// Mitsubishi GX Works2 project: 20190826   PLC: FX3U/FX3UC

PROGRAM MAIN
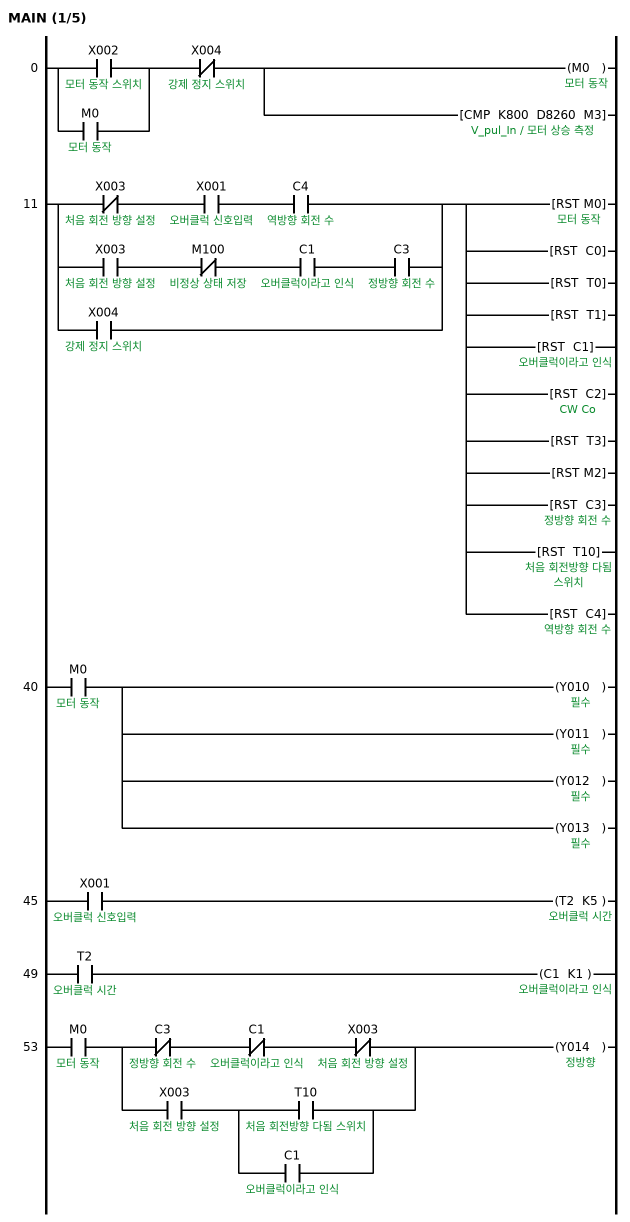
0     LD      X002  ; 모터 동작 스위치
      OR      M0  ; 모터 동작
      ANI     X004  ; 강제 정지 스위치
      OUT     M0  ; 모터 동작
      CMP     K800 D8260 M3  ; V_pul_In / 모터 상승 측정
11    LDI     X003  ; 처음 회전 방향 설정
      AND     X001  ; 오버클럭 신호입력
      AND     C4  ; 역방향 회전 수
      LD      X003  ; 처음 회전 방향 설정
      ANI     M100  ; 비정상 상태 저장
      AND     C1  ; 오버클럭이라고 인식
      AND     C3  ; 정방향 회전 수
      ORB
      OR      X004  ; 강제 정지 스위치
      RST     M0  ; 모터 동작
      RST     C0
      RST     T0
      RST     T1
      RST     C1  ; 오버클럭이라고 인식
      RST     C2  ; CW Co
      RST     T3
      RST     M2
      RST     C3  ; 정방향 회전 수
      RST     T10  ; 처음 회전방향 다됨 스위치
      RST     C4  ; 역방향 회전 수
40    LD      M0  ; 모터 동작
      OUT     Y010  ; 필수
      OUT     Y011  ; 필수
      OUT     Y012  ; 필수
      OUT     Y013  ; 필수
45    LD      X001  ; 오버클럭 신호입력
      OUT     T2 K5  ; 오버클럭 시간
49    LD      T2  ; 오버클럭 시간
      OUT     C1 K1  ; 오버클럭이라고 인식
53    LD      M0  ; 모터 동작
      LDI     C3  ; 정방향 회전 수
      ANI     C1  ; 오버클럭이라고 인식
      ANI     X003  ; 처음 회전 방향 설정
      LD      X003  ; 처음 회전 방향 설정
      LD      T10  ; 처음 회전방향 다됨 스위치
      OR      C1  ; 오버클럭이라고 인식
      ANB
      ORB
      ANB
      OUT     Y014  ; 정방향
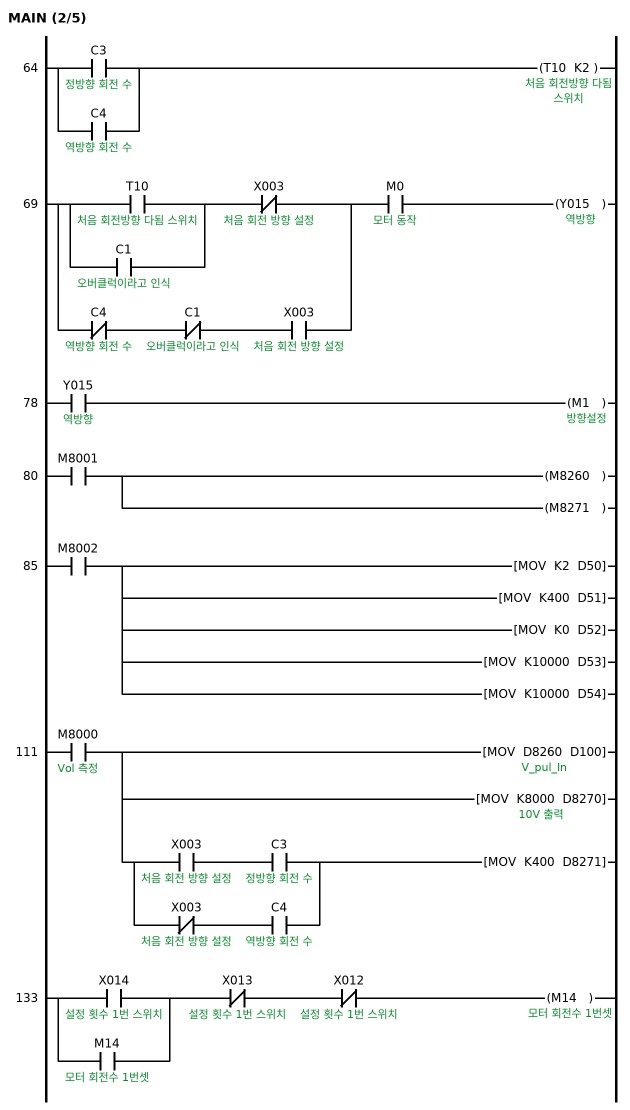
64    LD      C3  ; 정방향 회전 수
      OR      C4  ; 역방향 회전 수
      OUT     T10 K2  ; 처음 회전방향 다됨 스위치
69    LD      T10  ; 처음 회전방향 다됨 스위치
      OR      C1  ; 오버클럭이라고 인식
      ANI     X003  ; 처음 회전 방향 설정
      LDI     C4  ; 역방향 회전 수
      ANI     C1  ; 오버클럭이라고 인식
      AND     X003  ; 처음 회전 방향 설정
      ORB
      AND     M0  ; 모터 동작
      OUT     Y015  ; 역방향
78    LD      Y015  ; 역방향
      OUT     M1  ; 방향설정
80    LD      M8001
      OUT     M8260
      OUT     M8271
85    LD      M8002
      MOV     K2 D50
      MOV     K400 D51
      MOV     K0 D52
      MOV     K10000 D53
      MOV     K10000 D54
111   LD      M8000  ; Vol 측정
      MOV     D8260 D100
      MOV     K8000 D8270  ; 10V 출력
      LD      X003  ; 처음 회전 방향 설정
      AND     C3  ; 정방향 회전 수
      LDI     X003  ; 처음 회전 방향 설정
      AND     C4  ; 역방향 회전 수
      ORB
      ANB
      MOV     K400 D8271
133   LD      X014  ; 설정 횟수 1번 스위치
      OR      M14  ; 모터 회전수 1번셋
      ANI     X013  ; 설정 횟수 1번 스위치
      ANI     X012  ; 설정 횟수 1번 스위치
      OUT     M14  ; 모터 회전수 1번셋
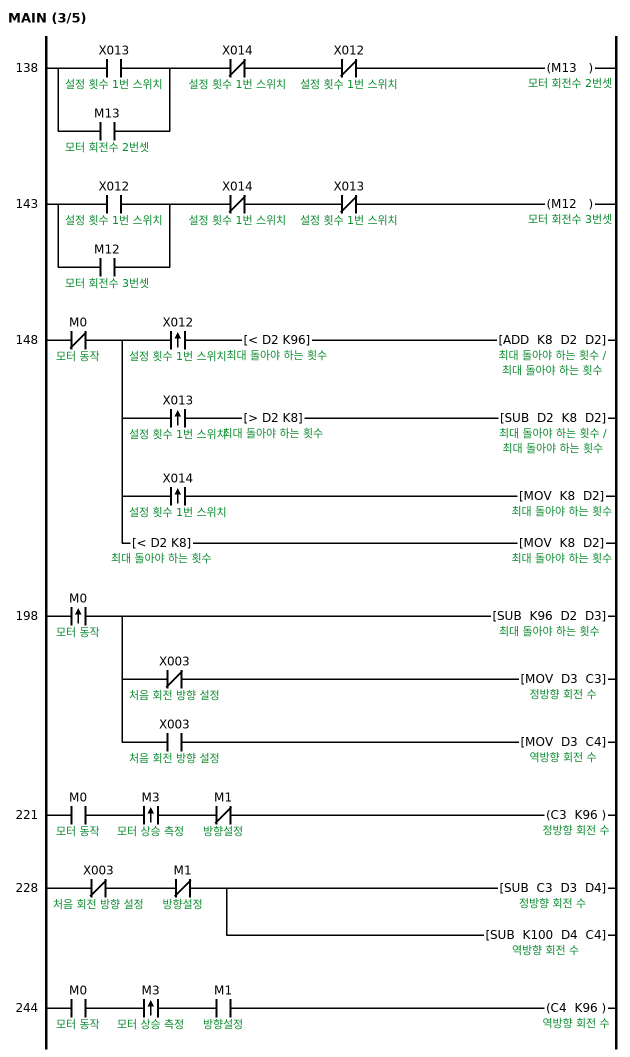
138   LD      X013  ; 설정 횟수 1번 스위치
      OR      M13  ; 모터 회전수 2번셋
      ANI     X014  ; 설정 횟수 1번 스위치
      ANI     X012  ; 설정 횟수 1번 스위치
      OUT     M13  ; 모터 회전수 2번셋
143   LD      X012  ; 설정 횟수 1번 스위치
      OR      M12  ; 모터 회전수 3번셋
      ANI     X014  ; 설정 횟수 1번 스위치
      ANI     X013  ; 설정 횟수 1번 스위치
      OUT     M12  ; 모터 회전수 3번셋
148   LDI     M0  ; 모터 동작
      MPS
      ANDP    X012  ; 설정 횟수 1번 스위치
      AND<    D2 K96  ; 최대 돌아야 하는 횟수
      ADD     K8 D2 D2
      MRD
      ANDP    X013  ; 설정 횟수 1번 스위치
      AND>    D2 K8  ; 최대 돌아야 하는 횟수
      SUB     D2 K8 D2
      MRD
      ANDP    X014  ; 설정 횟수 1번 스위치
      MOV     K8 D2
      MPP
      AND<    D2 K8  ; 최대 돌아야 하는 횟수
      MOV     K8 D2
198   LDP     M0  ; 모터 동작
      SUB     K96 D2 D3
      MPS
      ANI     X003  ; 처음 회전 방향 설정
      MOV     D3 C3
      MPP
      AND     X003  ; 처음 회전 방향 설정
      MOV     D3 C4
221   LD      M0  ; 모터 동작
      ANDP    M3  ; 모터 상승 측정
      ANI     M1  ; 방향설정
      OUT     C3 K96  ; 정방향 회전 수
228   LDI     X003  ; 처음 회전 방향 설정
      ANI     M1  ; 방향설정
      SUB     C3 D3 D4
      SUB     K100 D4 C4
244   LD      M0  ; 모터 동작
      ANDP    M3  ; 모터 상승 측정
      AND     M1  ; 방향설정
      OUT     C4 K96  ; 역방향 회전 수
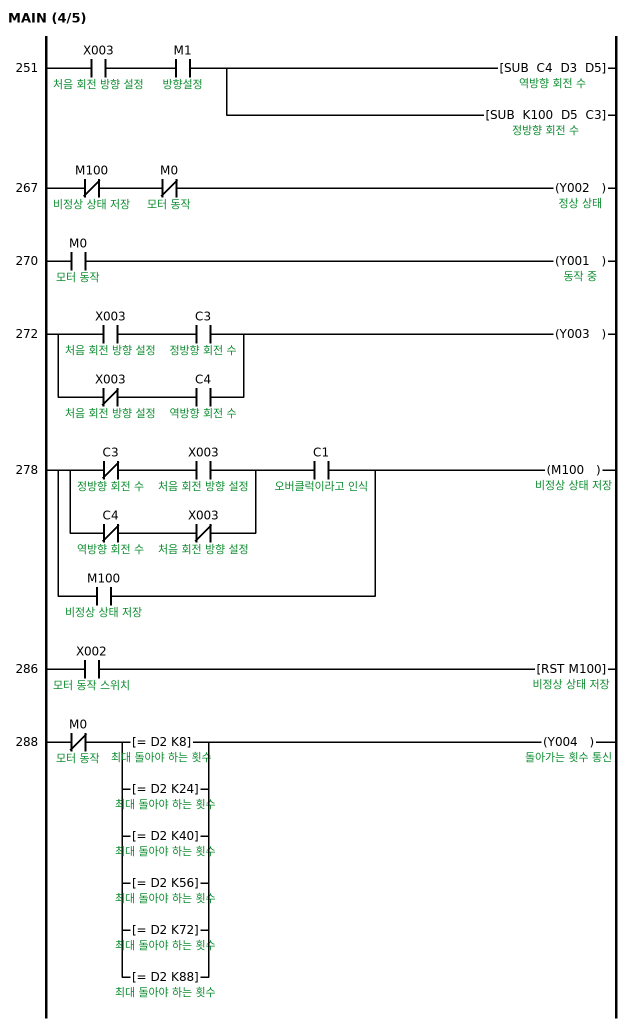
251   LD      X003  ; 처음 회전 방향 설정
      AND     M1  ; 방향설정
      SUB     C4 D3 D5
      SUB     K100 D5 C3
267   LDI     M100  ; 비정상 상태 저장
      ANI     M0  ; 모터 동작
      OUT     Y002  ; 정상 상태
270   LD      M0  ; 모터 동작
      OUT     Y001  ; 동작 중
272   LD      X003  ; 처음 회전 방향 설정
      AND     C3  ; 정방향 회전 수
      LDI     X003  ; 처음 회전 방향 설정
      AND     C4  ; 역방향 회전 수
      ORB
      OUT     Y003
278   LDI     C3  ; 정방향 회전 수
      AND     X003  ; 처음 회전 방향 설정
      LDI     C4  ; 역방향 회전 수
      ANI     X003  ; 처음 회전 방향 설정
      ORB
      AND     C1  ; 오버클럭이라고 인식
      OR      M100  ; 비정상 상태 저장
      OUT     M100  ; 비정상 상태 저장
286   LD      X002  ; 모터 동작 스위치
      RST     M100  ; 비정상 상태 저장
288   LDI     M0  ; 모터 동작
      LD=     D2 K8  ; 최대 돌아야 하는 횟수
      OR=     D2 K24  ; 최대 돌아야 하는 횟수
      OR=     D2 K40  ; 최대 돌아야 하는 횟수
      OR=     D2 K56  ; 최대 돌아야 하는 횟수
      OR=     D2 K72  ; 최대 돌아야 하는 횟수
      OR=     D2 K88  ; 최대 돌아야 하는 횟수
      ANB
      OUT     Y004  ; 돌아가는 횟수 통신
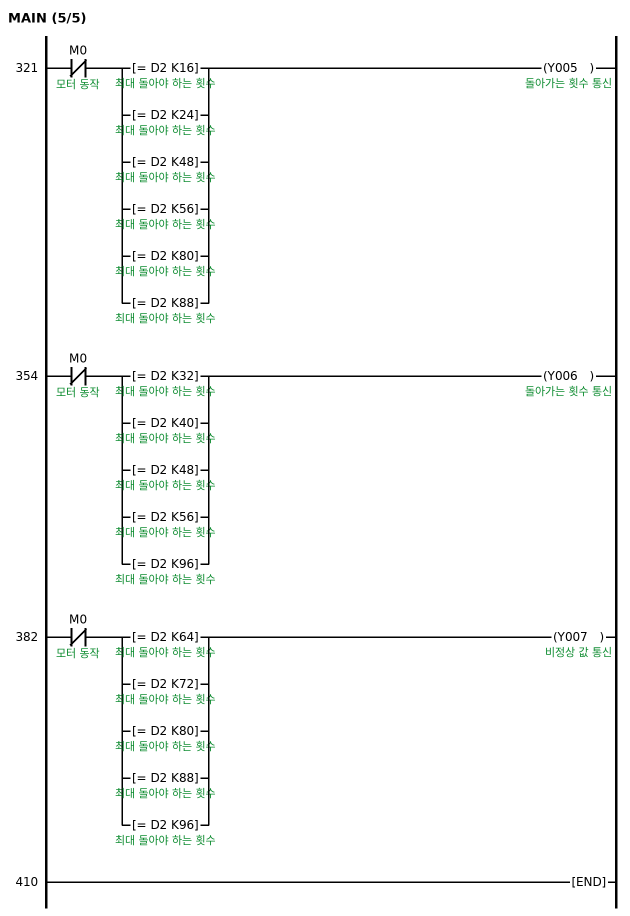
321   LDI     M0  ; 모터 동작
      LD=     D2 K16  ; 최대 돌아야 하는 횟수
      OR=     D2 K24  ; 최대 돌아야 하는 횟수
      OR=     D2 K48  ; 최대 돌아야 하는 횟수
      OR=     D2 K56  ; 최대 돌아야 하는 횟수
      OR=     D2 K80  ; 최대 돌아야 하는 횟수
      OR=     D2 K88  ; 최대 돌아야 하는 횟수
      ANB
      OUT     Y005  ; 돌아가는 횟수 통신
354   LDI     M0  ; 모터 동작
      LD=     D2 K32  ; 최대 돌아야 하는 횟수
      OR=     D2 K40  ; 최대 돌아야 하는 횟수
      OR=     D2 K48  ; 최대 돌아야 하는 횟수
      OR=     D2 K56  ; 최대 돌아야 하는 횟수
      OR=     D2 K96  ; 최대 돌아야 하는 횟수
      ANB
      OUT     Y006  ; 돌아가는 횟수 통신
382   LDI     M0  ; 모터 동작
      LD=     D2 K64  ; 최대 돌아야 하는 횟수
      OR=     D2 K72  ; 최대 돌아야 하는 횟수
      OR=     D2 K80  ; 최대 돌아야 하는 횟수
      OR=     D2 K88  ; 최대 돌아야 하는 횟수
      OR=     D2 K96  ; 최대 돌아야 하는 횟수
      ANB
      OUT     Y007  ; 비정상 값 통신
410   END
END_PROGRAM

// device comments not shown above
Y000  ; 비정상 상태
D1  ; 회전한 정방향 횟수 저장
D11  ; 역방향 횟수 저장
D12  ; 최대 돌아야하는 역방향 횟수
